{attribute 'linkalways'} 
{attribute 'no_explicit_call' := 'This FB is a CLASS and must be accessed using methods or properties'}
{attribute 'enable_dynamic_creation'}
FUNCTION_BLOCK FINAL GT_BYTE EXTENDS Node
VAR
	in1 : _BYTE(0);
	in2 : _BYTE(0);
	out : _BOOL(FALSE);
END_VAR

METHOD PUBLIC Clone : I_Node
VAR
	pNode : POINTER TO GT_BYTE;
END_VAR
pNode := __NEW(GT_BYTE);
Clone := pNode^;
END_METHOD

METHOD FB_init : BOOL
VAR_INPUT
	bInitRetains : BOOL; // if TRUE, the retain variables are initialized (warm start / cold start)
	bInCopyCode : BOOL;  // if TRUE, the instance afterwards gets moved into the copy code (online change)
END_VAR
AddInput('in1',THIS^.in1);
AddInput('in2',THIS^.in2);
AddOutput('out', THIS^.out);
END_METHOD

METHOD PROTECTED OnExecute
VAR
END_VAR
out.Value := in1.Value > in2.Value;
END_METHOD

END_FUNCTION_BLOCK

(* stored: Version 1.1.0.1, ProductVersion 3.1.4024.15
   POU GT_BYTE: Id {86228579-a63d-4678-af06-ab8cd78ff126}, SpecialFunc None
   Folder Constructor: Id {771d96db-13b9-47bc-aefd-28842d4b0963}
   Method Clone: Id {3cf3aa03-306c-4144-996c-9f4b641c7950}
   Method FB_init: Id {430d66f5-3f1d-48be-a07b-8e7aad6045df}
   Method OnExecute: Id {d44fa09c-98de-4a70-902d-9c00b471d1ac} *)
